// TIA Portal V16 export
// export: Created 2021-10-07T09:38:24.5980071Z, ExportSetting None, DisplayName Totally Integrated Automation Portal, DisplayVersion V16 Update 4, DisplayName TIA Portal Version Control Interface, DisplayVersion V16 Update 2, DisplayName TIA Portal Openness, DisplayVersion V16 Update 4, DisplayName SINAMICS Startdrive Advanced, DisplayVersion V16 Update 5, DisplayName SINAMICS Startdrive G130, G150, S120, S150, SINAMICS MV, S210, DisplayVersion V16 Update 5, DisplayName SINAMICS Startdrive G110M, G120, G120C, G120D, G120P, G115D, DisplayVersion V16 Update 5, DisplayName STEP 7 Professional, DisplayVersion V16 Update 4, DisplayName STEP 7 Safety, DisplayVersion V16, DisplayName WinCC Advanced, DisplayVersion V16 Update 4
FUNCTION "fcTest" : Void   // FC1, LAD
{ S7_Optimized_Access := 'TRUE' }
// stored: SetENOAutomatically false
   VAR_INPUT
      CoolInput : Real;
      HotInput : UDInt;
   END_VAR
   VAR_OUTPUT
      ColdOutput : Word;
      HotOutput : Struct
         Hot1 : CONN_ANY;
         Hot2 : Date_And_Time;
         Hot3 : Array[0..9] of Char;
      END_STRUCT;
   END_VAR
   VAR_IN_OUT
      ColdInOut : IEC_TIMER;
      HotInOut : IEC_COUNTER;
   END_VAR
   VAR_TEMP
      tCold : "UDT_Test";
      tHot : DInt;
   END_VAR
   VAR CONSTANT
      COLD_CONSTANT : Int;
      HOT_CONSTANT : Real;
   END_VAR
BEGIN

REGION Network 1: Segmento1!
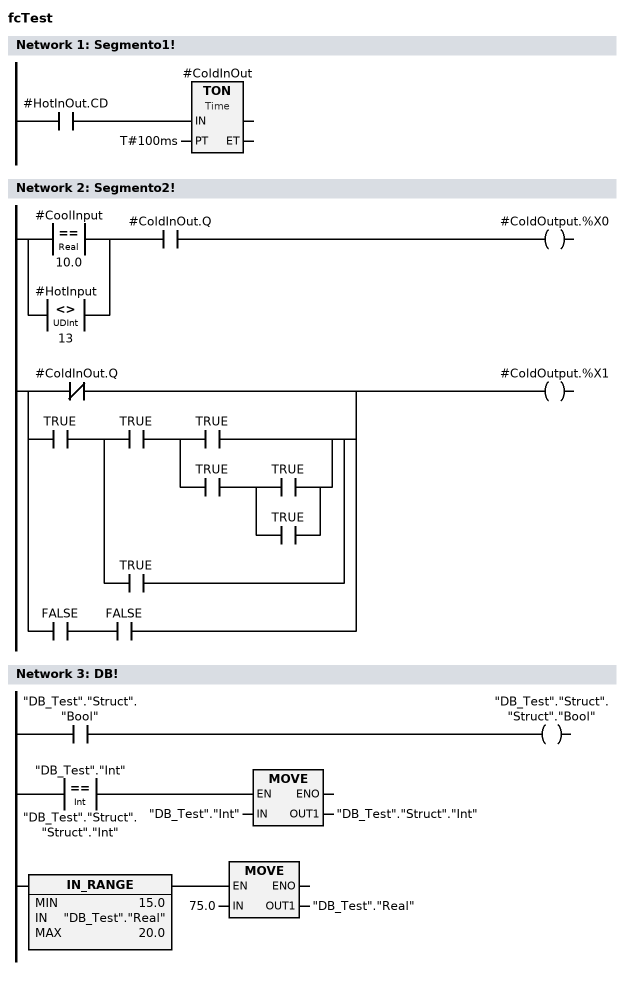
   RUNG wire#powerrail
      Contact( #HotInOut.CD )
      { S7_Templates := "time_type := Time" } #ColdInOut.TON(pt := T#100ms, et =>)
   END_RUNG
   // the same network as SCL:
   #ColdInOut.TON(IN := #HotInOut.CD, PT := T#100ms);
END_REGION

REGION Network 2: Segmento2!
   RUNG wire#powerrail
      { S7_Templates := "SrcType := Real" } EQ_Contact(in1 := #CoolInput, in2 := 10.0)
      wire#w1
      Contact( #ColdInOut.Q )
      Coil( #ColdOutput.%X0 )
   END_RUNG
   RUNG wire#powerrail
      { S7_Templates := "SrcType := UDInt" } NE_Contact(in1 := #HotInput, in2 := 13)
   END_RUNG wire#w1
   RUNG wire#powerrail
      I_Contact( #ColdInOut.Q )
      wire#w2
      Coil( #ColdOutput.%X1 )
   END_RUNG
   RUNG wire#powerrail
      Contact( TRUE )
      wire#w3
      Contact( TRUE )
      wire#w4
      Contact( TRUE )
   END_RUNG wire#w2
   RUNG wire#w4
      Contact( TRUE )
      wire#w5
      Contact( TRUE )
   END_RUNG wire#w2
   RUNG wire#w5
      Contact( TRUE )
   END_RUNG wire#w2
   RUNG wire#w3
      Contact( TRUE )
   END_RUNG wire#w2
   RUNG wire#powerrail
      Contact( FALSE )
      Contact( FALSE )
   END_RUNG wire#w2
   // the same network as SCL:
   #ColdOutput.%X0 := ((#CoolInput = 10.0) OR (#HotInput <> 13)) AND #ColdInOut.Q;
   #ColdOutput.%X1 := NOT #ColdInOut.Q OR (TRUE AND ((TRUE AND (TRUE OR (TRUE AND (TRUE OR TRUE)))) OR TRUE)) OR (FALSE AND FALSE);
END_REGION

REGION Network 3: DB!
   RUNG wire#powerrail
      Contact( "DB_Test"."Struct"."Bool" )
      Coil( "DB_Test"."Struct"."Struct"."Bool" )
   END_RUNG
   RUNG wire#powerrail
      { S7_Templates := "SrcType := Int" } EQ_Contact(in1 := "DB_Test"."Int", in2 := "DB_Test"."Struct"."Struct"."Int")
      Move(in := "DB_Test"."Int", out1 => "DB_Test"."Struct"."Int")
   END_RUNG
   RUNG wire#powerrail
      { S7_Templates := "SrcType := Real" } InRange(min := 15.0, in := "DB_Test"."Real", max := 20.0)
      Move(in := 75.0, out1 => "DB_Test"."Real")
   END_RUNG
   // the same network as SCL:
   "DB_Test"."Struct"."Struct"."Bool" := "DB_Test"."Struct"."Bool";
   IF "DB_Test"."Int" = "DB_Test"."Struct"."Struct"."Int" THEN
       "DB_Test"."Struct"."Int" := "DB_Test"."Int";
   END_IF;
   IF (15.0 <= "DB_Test"."Real") AND ("DB_Test"."Real" <= 20.0) THEN "DB_Test"."Real" := 75.0; END_IF;
END_REGION

REGION Network 4 (SCL): SCL!
   IF #CoolInput <> 100 THEN
       #HotInOut.CD := FALSE;
   END_IF;
END_REGION
END_FUNCTION
